(* IEC 61131-3 sources: IRT/Program, 4 files *)

(* ---- CalcD.fb ---- *)
FUNCTION_BLOCK CalcD
VAR_INPUT
	input 			:	REAL;
	KD				:	REAL;
	error			:	REAL;
END_VAR

VAR_OUTPUT
	output 			:	REAL;
END_VAR

VAR
	init			:	BOOL;
	currentTime		:	DWORD;
	lastTime		:	DWORD;
	timeDiff		:	REAL;
	lastError		:	REAL;
END_VAR

currenttime := TIME_TO_DWORD(Time());
timeDiff := DWORD_TO_REAL(currentTime - lastTime);

IF NOT init THEN
	init := TRUE;
	lastError := error;
ELSIF timeDiff > 0.0 THEN
	output := KD * ((error / lastError) / timeDiff);
	lastError := error;
ELSE
	output := 0.0;
END_IF
lastTime := currenttime

(* ---- CalcI.fb ---- *)
FUNCTION_BLOCK CalcI
VAR_INPUT
	input 		:	REAL;
	KI			:	REAL;
	outMin		:	REAL; // Minimum outputvalue
	outMax		:	REAL; // Maximum outputvalue
	error		:	REAL;
END_VAR

VAR_OUTPUT
	limit		:	BOOL;
	output 		:	REAL;
END_VAR

VAR
	oldValue	:	REAL;
	init		:	BOOL;
	currentTime	:	DWORD;
	lastTime	:	DWORD;
	timeDiff	:	REAL;

	errorSum	:	REAL;
END_VAR

currentTime := TIME_TO_DWORD(Time()); // to seconds
timeDiff := DWORD_TO_REAL(currentTime - lastTime); // Calculate the timedifference between now and last calculation
// Integrator calculations
IF NOT init THEN
	init := TRUE;
	oldValue := input;
ELSIF timeDiff > 0.0 THEN
	errorSum := errorSum + (error * timeDiff);
	output := KI * errorSum;
END_IF

IF output > outMax THEN
	errorSum := outMax * (1/KI);
	limit := TRUE;
ELSIF output <= outMin THEN
	output := outMin;
	errorSum := outMin * (1/KI);
	limit := TRUE;
ELSE
	limit := FALSE;
END_IF

lastTime := currentTime;

(* ---- PID.fb ---- *)
FUNCTION_BLOCK pid

VAR_INPUT
	KP	:	REAL;
	KI	:	REAL;
	KD	:	REAL;

	IlimMin		:	REAL; // Lower limit of the integrator
	IlimMax		:	REAL; // Upper limit of the integrator
	setPoint	:	REAL;
	in 			:	REAL;
END_VAR

VAR_OUTPUT
	limit		:	BOOL; // Limit of the PID (active/inactive)
	Y			:	REAL; // Output of the PID
END_VAR

VAR
	Dcalc		:	CalcD;
	Icalc		:	CalcI;

	error		:	REAL;
END_VAR

error := setPoint - in;
Icalc(input := in, KI := KI, outMin := IlimMin, outMax := IlimMax, error := error);
Dcalc(input := in, Kd := KD, error := error);

Y := KP * error + Icalc.output + Dcalc.output;

(* ---- PLC_PRG.st ---- *)
PROGRAM PLC_PRG
VAR
	pid			:	PID;

	Lmin		:	REAL := -2;
	Lmax		:	REAL := 2;
	setPoint	:	REAL := 5.0;

	kP			:	REAL := 1.5;
	kI			:	REAL := 0.1;
	Kd			:	REAL := 2.5;
END_VAR

pid(KP := kP, KI := kI, KD := kD, IlimMin := Lmin, IlimMax := Lmax, setpoint := setpoint, in := Tank.METER_LEVEL);

IF pid.Y > 0 THEN
	Tank.VALVE_FILL := pid.Y;
	Tank.VALVE_DISCHARGE := 0;
ELSIF pid.Y < 0 THEN
	Tank.VALVE_DISCHARGE := (pid.Y * -1);
	Tank.VALVE_FILL := 0;
ELSE
	Tank.VALVE_DISCHARGE := 0;
	Tank.VALVE_FILL := 0;
END_IF
